FUNCTION_BLOCK FB_Syntax_OOP
VAR
    _nInternal : INT;
END_VAR

_nInternal := _nInternal + 1;

METHOD M_Increment : BOOL
VAR_INPUT
    nDelta : INT;
END_VAR
_nInternal  := _nInternal + nDelta;
M_Increment := TRUE;
END_METHOD

PROPERTY P_Count : INT
GET
P_Count := _nInternal;
END_GET
END_PROPERTY

END_FUNCTION_BLOCK

(* stored: Version 1.1.0.1, ProductVersion 3.1.4024.16
   POU FB_Syntax_OOP: Id {0306bcb6-6e06-4540-86d2-51a4ca547d0a}, SpecialFunc None
   Method M_Increment: Id {d955123b-591e-457d-b44f-26a5e9f23c76}
   Property P_Count: Id {ab96ac50-24ec-492b-9f0c-0cc05dda2ea8}
   Get Get: Id {e431525a-4cb6-4194-916c-e59e954fa028} *)
